% RSLogix 500 project VA116_TR_D.RSS, saved by version 7.10.00.09 %
PROJECT "VA116"    % processor: SLC 500, 1747-L532; 601760_CO2 %

PROGRAM FILES
  LAD 2 "601760_CO2"  66 rungs
  LAD 3 "INIT_ZAPN"  24 rungs
  LAD 4 "CASOVACE"  76 rungs
  LAD 5 "DIAGN_SPOL"  16 rungs
  LAD 6 "DIAGN_AUT"  98 rungs
  LAD 7 "DIAGN_K_VP"  28 rungs
  LAD 8 "HYDR_AGREG"  13 rungs
  LAD 9 "VODA_POHON"  16 rungs
  LAD 10 "REZIM_SER"  50 rungs
  LAD 11 "REZIM_RUC"  66 rungs
  LAD 12 "REZIM_VP"  18 rungs
  LAD 13 "REZIM_AUT"  28 rungs
  LAD 14 "REZIM_NULA"  6 rungs
  LAD 15 "STARTSTOP"  28 rungs
  LAD 16 "ZAKL_MECH"  92 rungs
  LAD 17 "KOPYTO_SOL"  22 rungs
  LAD 18 "HLAVA_SOLO"  23 rungs
  LAD 19 "KOPY_HLAVA"  37 rungs
  LAD 20 "STABILIZ"  24 rungs
  LAD 21 "ODDEL_IMP"  19 rungs
  LAD 22 "ODDEL_RS"  29 rungs
  LAD 23 "PODPUR_VZD"  17 rungs
  LAD 24 "VYFUK_TRN"  33 rungs
  LAD 25 "CO2"  8 rungs
  LAD 26 "VYSTUPY"  81 rungs
  LAD 27 "REC_ARCHIV"  4 rungs
  LAD 28 "REC_SAVE"  3 rungs
  LAD 29 "REC_LOAD"  4 rungs
  LAD 30 "REG_TEPLOT"  149 rungs

DATA FILES
  O0   38 elements
  I1   36 elements
  S2   83 elements
  B3   2 elements
  T4   82 elements
  C5   6 elements
  R6   1 elements
  N7   98 elements
  F8 FLOAT  10 elements
  N9   12 elements
  N10   256 elements
  N11   256 elements
  N12 N12  240 elements
  N13   255 elements
  N14   240 elements
  N15   240 elements

LADDER 2 "601760_CO2"
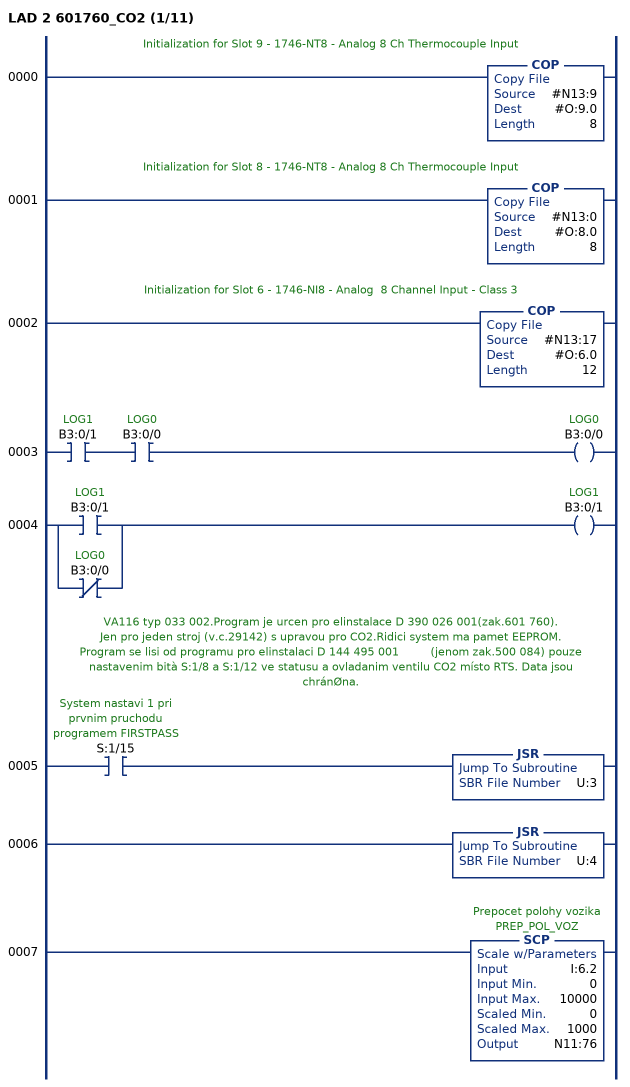
% Rung: 0 %
% Initialization for Slot 9 - 1746-NT8 - Analog 8 Ch Thermocouple Input %
SOR COP #N13:9 #O:9.0 8 EOR
% Rung: 1 %
% Initialization for Slot 8 - 1746-NT8 - Analog 8 Ch Thermocouple Input %
SOR COP #N13:0 #O:8.0 8 EOR
% Rung: 2 %
% Initialization for Slot 6 - 1746-NI8 - Analog  8 Channel Input - Class 3 %
SOR COP #N13:17 #O:6.0 12 EOR
% Rung: 3 %
SOR XIC B3:0/1 XIC B3:0/0 OTE B3:0/0 EOR
%   B3:0/1  LOG1 %
%   B3:0/0  LOG0 %
% Rung: 4 %
SOR BST XIC B3:0/1 NXB XIO B3:0/0 BND OTE B3:0/1 EOR
%   B3:0/1  LOG1 %
%   B3:0/0  LOG0 %
% Rung: 5 %
% VA116 typ 033 002.Program je urcen pro elinstalace D 390 026 001(zak.601 760).
% Jen pro jeden stroj (v.c.29142) s upravou pro CO2.Ridici system ma pamet EEPROM. Program se lisi od programu pro elinstalaci D 144 495 001         (jenom zak.500 084) pouze nastavenim bità S:1/8 a S:1/12 ve statusu a ovladanim ventilu CO2 místo RTS. Data jsou chránØna. %
SOR XIC S:1/15 JSR U:3 EOR
%   S:1/15  FIRSTPASS  "System nastavi 1 pri prvnim pruchodu programem" %
%   JSR U:3  "Iniciali- zace po zapnuti ridiciho systemu" %
% Rung: 6 %
SOR JSR U:4 EOR
%   JSR U:4  "Casovace, citace" %
% Rung: 7 %
SOR SCP I:6.2 0 10000 0 1000 N11:76 EOR
%   I:6.2  POL_VOZIKA  "Poloha vozika" %
%   N11:76  PREP_POL_VOZ  "Prepocet polohy vozika" %

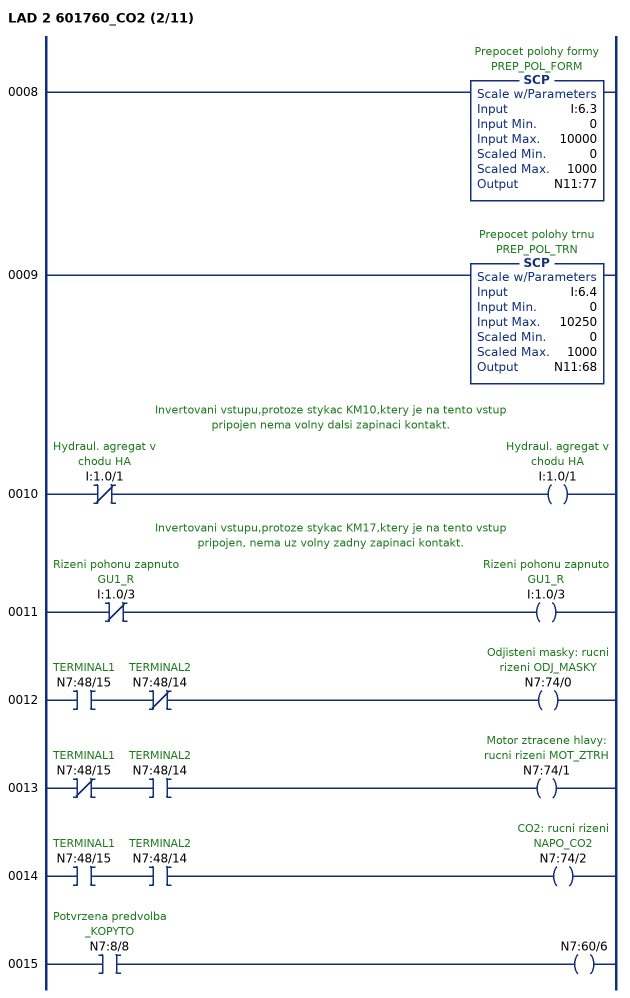
% Rung: 8 %
SOR SCP I:6.3 0 10000 0 1000 N11:77 EOR
%   I:6.3  POL_FORMY  "Poloha formy" %
%   N11:77  PREP_POL_FORM  "Prepocet polohy formy" %
% Rung: 9 %
SOR SCP I:6.4 0 10250 0 1000 N11:68 EOR
%   I:6.4  POL_VYF_TRNU  "Poloha vyfukovaciho trnu" %
%   N11:68  PREP_POL_TRN  "Prepocet polohy trnu" %
% Rung: 10 %
%         Invertovani vstupu,protoze stykac KM10,ktery je na tento vstup
%         pripojen nema volny dalsi zapinaci kontakt. %
SOR XIO I:1.0/1 OTE I:1.0/1 EOR
%   I:1.0/1  HA  "Hydraul. agregat v chodu" %
% Rung: 11 %
%          Invertovani vstupu,protoze stykac KM17,ktery je na tento vstup
%          pripojen, nema uz volny zadny zapinaci kontakt. %
SOR XIO I:1.0/3 OTE I:1.0/3 EOR
%   I:1.0/3  GU1_R  "Rizeni pohonu zapnuto" %
% Rung: 12 %
SOR XIC N7:48/15 XIO N7:48/14 OTE N7:74/0 EOR
%   N7:48/15  TERMINAL1 %
%   N7:48/14  TERMINAL2 %
%   N7:74/0  ODJ_MASKY  "Odjisteni masky: rucni rizeni" %
% Rung: 13 %
SOR XIO N7:48/15 XIC N7:48/14 OTE N7:74/1 EOR
%   N7:48/15  TERMINAL1 %
%   N7:48/14  TERMINAL2 %
%   N7:74/1  MOT_ZTRH  "Motor ztracene hlavy: rucni rizeni" %
% Rung: 14 %
SOR XIC N7:48/15 XIC N7:48/14 OTE N7:74/2 EOR
%   N7:48/15  TERMINAL1 %
%   N7:48/14  TERMINAL2 %
%   N7:74/2  NAPO_CO2  "CO2: rucni rizeni" %
% Rung: 15 %
SOR XIC N7:8/8 OTE N7:60/6 EOR
%   N7:8/8  _KOPYTO  "Potvrzena predvolba" %

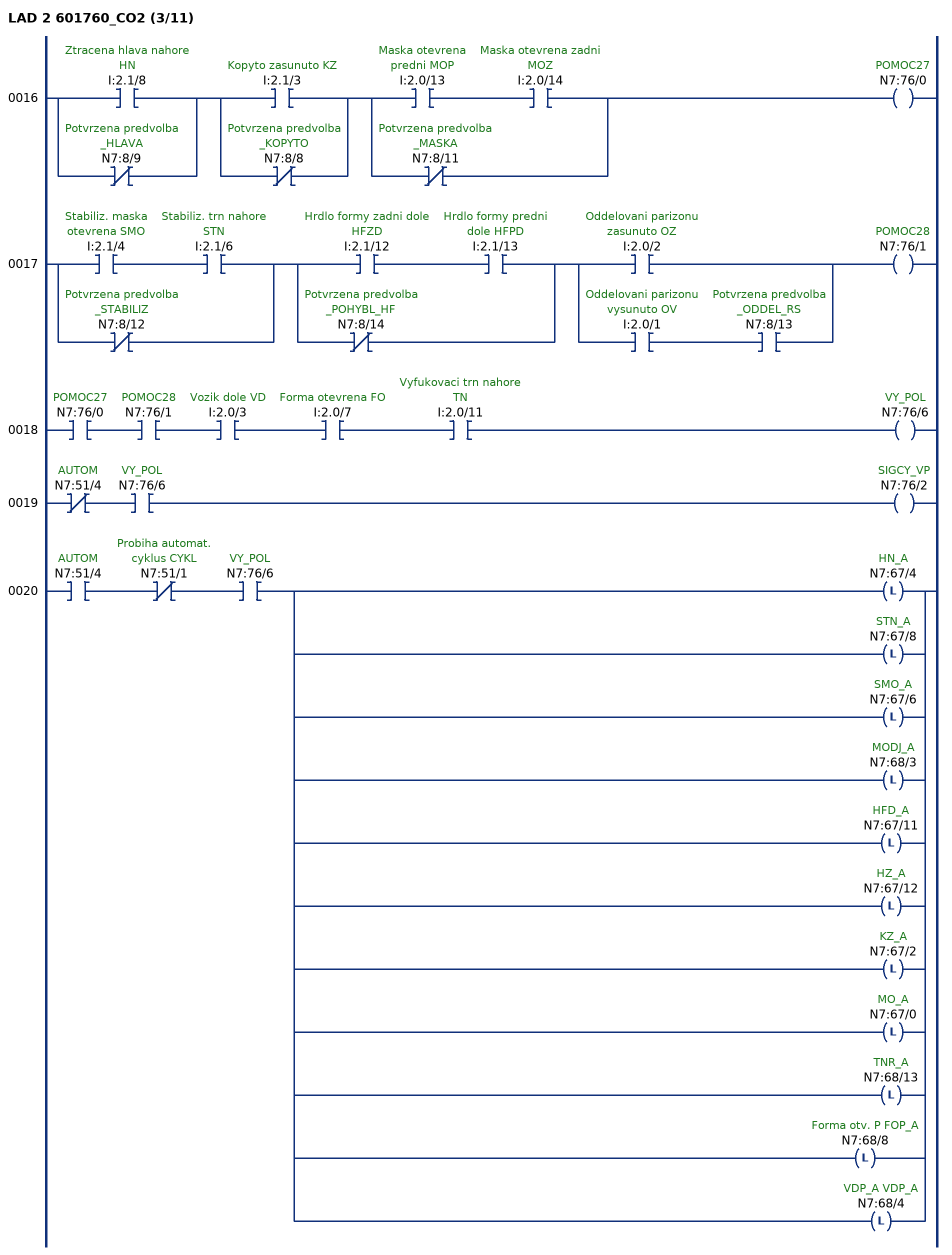
% Rung: 16 %
SOR BST XIC I:2.1/8 NXB XIO N7:8/9 BND BST XIC I:2.1/3 NXB XIO N7:8/8 BND BST XIC I:2.0/13 XIC I:2.0/14 NXB XIO N7:8/11 BND OTE N7:76/0 EOR
%   I:2.1/8  HN  "Ztracena hlava nahore" %
%   N7:8/9  _HLAVA  "Potvrzena predvolba" %
%   I:2.1/3  KZ  "Kopyto zasunuto" %
%   N7:8/8  _KOPYTO  "Potvrzena predvolba" %
%   I:2.0/13  MOP  "Maska otevrena predni" %
%   I:2.0/14  MOZ  "Maska otevrena zadni" %
%   N7:8/11  _MASKA  "Potvrzena predvolba" %
%   N7:76/0  POMOC27 %
% Rung: 17 %
SOR BST XIC I:2.1/4 XIC I:2.1/6 NXB XIO N7:8/12 BND BST XIC I:2.1/12 XIC I:2.1/13 NXB XIO N7:8/14 BND BST XIC I:2.0/2 NXB XIC I:2.0/1 XIC N7:8/13 BND OTE N7:76/1 EOR
%   I:2.1/4  SMO  "Stabiliz. maska otevrena" %
%   I:2.1/6  STN  "Stabiliz. trn nahore" %
%   N7:8/12  _STABILIZ  "Potvrzena predvolba" %
%   I:2.1/12  HFZD  "Hrdlo formy zadni dole" %
%   I:2.1/13  HFPD  "Hrdlo formy predni dole" %
%   N7:8/14  _POHYBL_HF  "Potvrzena predvolba" %
%   I:2.0/2  OZ  "Oddelovani parizonu zasunuto" %
%   I:2.0/1  OV  "Oddelovani parizonu vysunuto" %
%   N7:8/13  _ODDEL_RS  "Potvrzena predvolba" %
%   N7:76/1  POMOC28 %
% Rung: 18 %
SOR XIC N7:76/0 XIC N7:76/1 XIC I:2.0/3 XIC I:2.0/7 XIC I:2.0/11 OTE N7:76/6 EOR
%   N7:76/0  POMOC27 %
%   N7:76/1  POMOC28 %
%   I:2.0/3  VD  "Vozik dole" %
%   I:2.0/7  FO  "Forma otevrena" %
%   I:2.0/11  TN  "Vyfukovaci trn nahore" %
%   N7:76/6  VY_POL %
% Rung: 19 %
SOR XIO N7:51/4 XIC N7:76/6 OTE N7:76/2 EOR
%   N7:51/4  AUTOM %
%   N7:76/6  VY_POL %
%   N7:76/2  SIGCY_VP %
% Rung: 20 %
SOR XIC N7:51/4 XIO N7:51/1 XIC N7:76/6 BST OTL N7:67/4 NXB OTL N7:67/8 NXB OTL N7:67/6 NXB OTL N7:68/3 NXB OTL N7:67/11 NXB OTL N7:67/12 NXB OTL N7:67/2 NXB OTL N7:67/0 NXB OTL N7:68/13 NXB OTL N7:68/8 NXB OTL N7:68/4 BND EOR
%   N7:51/4  AUTOM %
%   N7:51/1  CYKL  "Probiha automat. cyklus" %
%   N7:76/6  VY_POL %
%   N7:67/4  HN_A %
%   N7:67/8  STN_A %
%   N7:67/6  SMO_A %
%   N7:68/3  MODJ_A %
%   N7:67/11  HFD_A %
%   N7:67/12  HZ_A %
%   N7:67/2  KZ_A %
%   N7:67/0  MO_A %
%   N7:68/13  TNR_A %
%   N7:68/8  FOP_A  "Forma otv. P" %
%   N7:68/4  VDP_A  "VDP_A" %

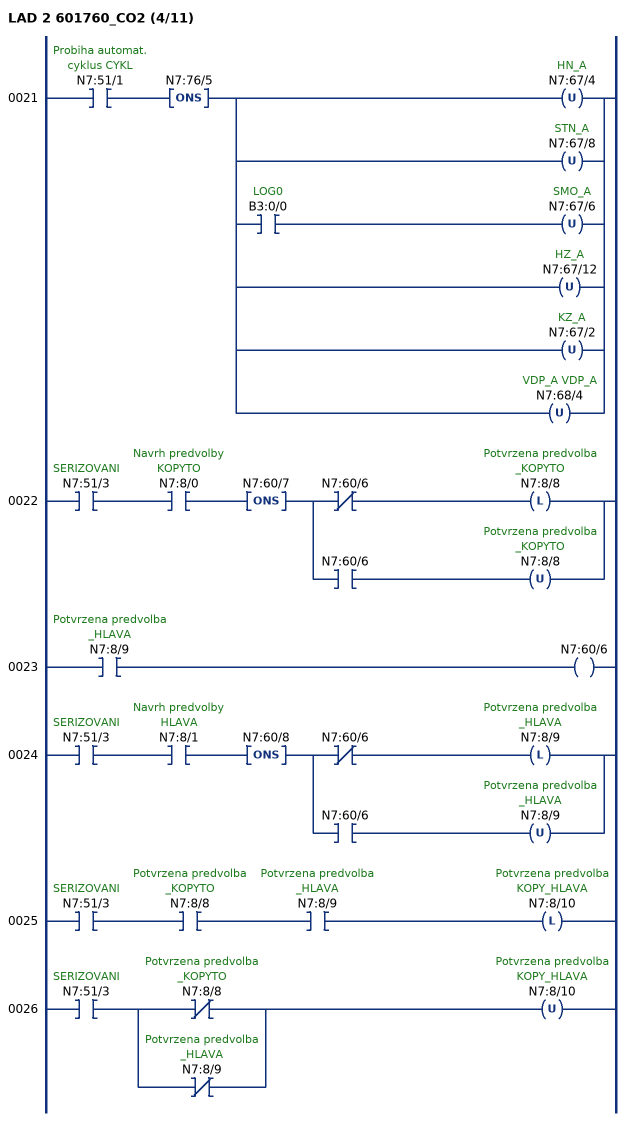
% Rung: 21 %
SOR XIC N7:51/1 OSR N7:76/5 BST OTU N7:67/4 NXB OTU N7:67/8 NXB XIC B3:0/0 OTU N7:67/6 NXB OTU N7:67/12 NXB OTU N7:67/2 NXB OTU N7:68/4 BND EOR
%   N7:51/1  CYKL  "Probiha automat. cyklus" %
%   N7:67/4  HN_A %
%   N7:67/8  STN_A %
%   B3:0/0  LOG0 %
%   N7:67/6  SMO_A %
%   N7:67/12  HZ_A %
%   N7:67/2  KZ_A %
%   N7:68/4  VDP_A  "VDP_A" %
% Rung: 22 %
SOR XIC N7:51/3 XIC N7:8/0 OSR N7:60/7 BST XIO N7:60/6 OTL N7:8/8 NXB XIC N7:60/6 OTU N7:8/8 BND EOR
%   N7:51/3  SERIZOVANI %
%   N7:8/0  KOPYTO  "Navrh predvolby" %
%   N7:8/8  _KOPYTO  "Potvrzena predvolba" %
% Rung: 23 %
SOR XIC N7:8/9 OTE N7:60/6 EOR
%   N7:8/9  _HLAVA  "Potvrzena predvolba" %
% Rung: 24 %
SOR XIC N7:51/3 XIC N7:8/1 OSR N7:60/8 BST XIO N7:60/6 OTL N7:8/9 NXB XIC N7:60/6 OTU N7:8/9 BND EOR
%   N7:51/3  SERIZOVANI %
%   N7:8/1  HLAVA  "Navrh predvolby" %
%   N7:8/9  _HLAVA  "Potvrzena predvolba" %
% Rung: 25 %
SOR XIC N7:51/3 XIC N7:8/8 XIC N7:8/9 OTL N7:8/10 EOR
%   N7:51/3  SERIZOVANI %
%   N7:8/8  _KOPYTO  "Potvrzena predvolba" %
%   N7:8/9  _HLAVA  "Potvrzena predvolba" %
%   N7:8/10  KOPY_HLAVA  "Potvrzena predvolba" %
% Rung: 26 %
SOR XIC N7:51/3 BST XIO N7:8/8 NXB XIO N7:8/9 BND OTU N7:8/10 EOR
%   N7:51/3  SERIZOVANI %
%   N7:8/8  _KOPYTO  "Potvrzena predvolba" %
%   N7:8/9  _HLAVA  "Potvrzena predvolba" %
%   N7:8/10  KOPY_HLAVA  "Potvrzena predvolba" %

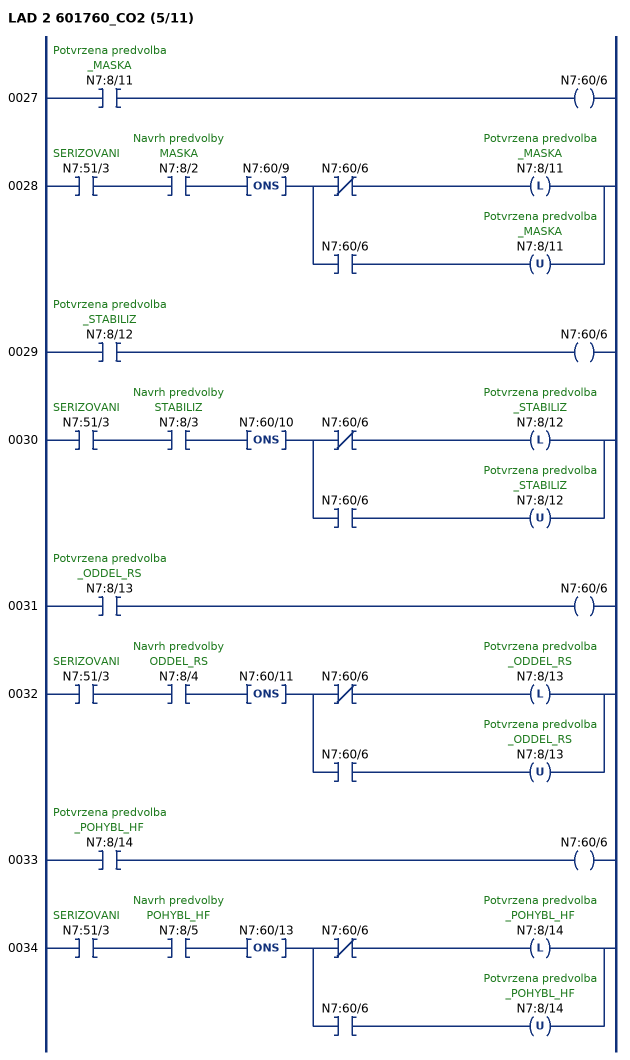
% Rung: 27 %
SOR XIC N7:8/11 OTE N7:60/6 EOR
%   N7:8/11  _MASKA  "Potvrzena predvolba" %
% Rung: 28 %
SOR XIC N7:51/3 XIC N7:8/2 OSR N7:60/9 BST XIO N7:60/6 OTL N7:8/11 NXB XIC N7:60/6 OTU N7:8/11 BND EOR
%   N7:51/3  SERIZOVANI %
%   N7:8/2  MASKA  "Navrh predvolby" %
%   N7:8/11  _MASKA  "Potvrzena predvolba" %
% Rung: 29 %
SOR XIC N7:8/12 OTE N7:60/6 EOR
%   N7:8/12  _STABILIZ  "Potvrzena predvolba" %
% Rung: 30 %
SOR XIC N7:51/3 XIC N7:8/3 OSR N7:60/10 BST XIO N7:60/6 OTL N7:8/12 NXB XIC N7:60/6 OTU N7:8/12 BND EOR
%   N7:51/3  SERIZOVANI %
%   N7:8/3  STABILIZ  "Navrh predvolby" %
%   N7:8/12  _STABILIZ  "Potvrzena predvolba" %
% Rung: 31 %
SOR XIC N7:8/13 OTE N7:60/6 EOR
%   N7:8/13  _ODDEL_RS  "Potvrzena predvolba" %
% Rung: 32 %
SOR XIC N7:51/3 XIC N7:8/4 OSR N7:60/11 BST XIO N7:60/6 OTL N7:8/13 NXB XIC N7:60/6 OTU N7:8/13 BND EOR
%   N7:51/3  SERIZOVANI %
%   N7:8/4  ODDEL_RS  "Navrh predvolby" %
%   N7:8/13  _ODDEL_RS  "Potvrzena predvolba" %
% Rung: 33 %
SOR XIC N7:8/14 OTE N7:60/6 EOR
%   N7:8/14  _POHYBL_HF  "Potvrzena predvolba" %
% Rung: 34 %
SOR XIC N7:51/3 XIC N7:8/5 OSR N7:60/13 BST XIO N7:60/6 OTL N7:8/14 NXB XIC N7:60/6 OTU N7:8/14 BND EOR
%   N7:51/3  SERIZOVANI %
%   N7:8/5  POHYBL_HF  "Navrh predvolby" %
%   N7:8/14  _POHYBL_HF  "Potvrzena predvolba" %

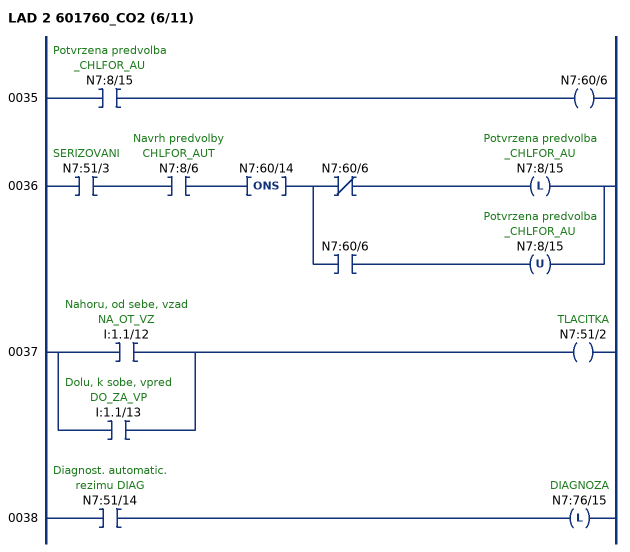
% Rung: 35 %
SOR XIC N7:8/15 OTE N7:60/6 EOR
%   N7:8/15  _CHLFOR_AU  "Potvrzena predvolba" %
% Rung: 36 %
SOR XIC N7:51/3 XIC N7:8/6 OSR N7:60/14 BST XIO N7:60/6 OTL N7:8/15 NXB XIC N7:60/6 OTU N7:8/15 BND EOR
%   N7:51/3  SERIZOVANI %
%   N7:8/6  CHLFOR_AUT  "Navrh predvolby" %
%   N7:8/15  _CHLFOR_AU  "Potvrzena predvolba" %
% Rung: 37 %
SOR BST XIC I:1.1/12 NXB XIC I:1.1/13 BND OTE N7:51/2 EOR
%   I:1.1/12  NA_OT_VZ  "Nahoru, od sebe, vzad" %
%   I:1.1/13  DO_ZA_VP  "Dolu, k sobe, vpred" %
%   N7:51/2  TLACITKA %
% Rung: 38 %
SOR XIC N7:51/14 OTL N7:76/15 EOR
%   N7:51/14  DIAG  "Diagnost. automatic. rezimu" %
%   N7:76/15  DIAGNOZA %

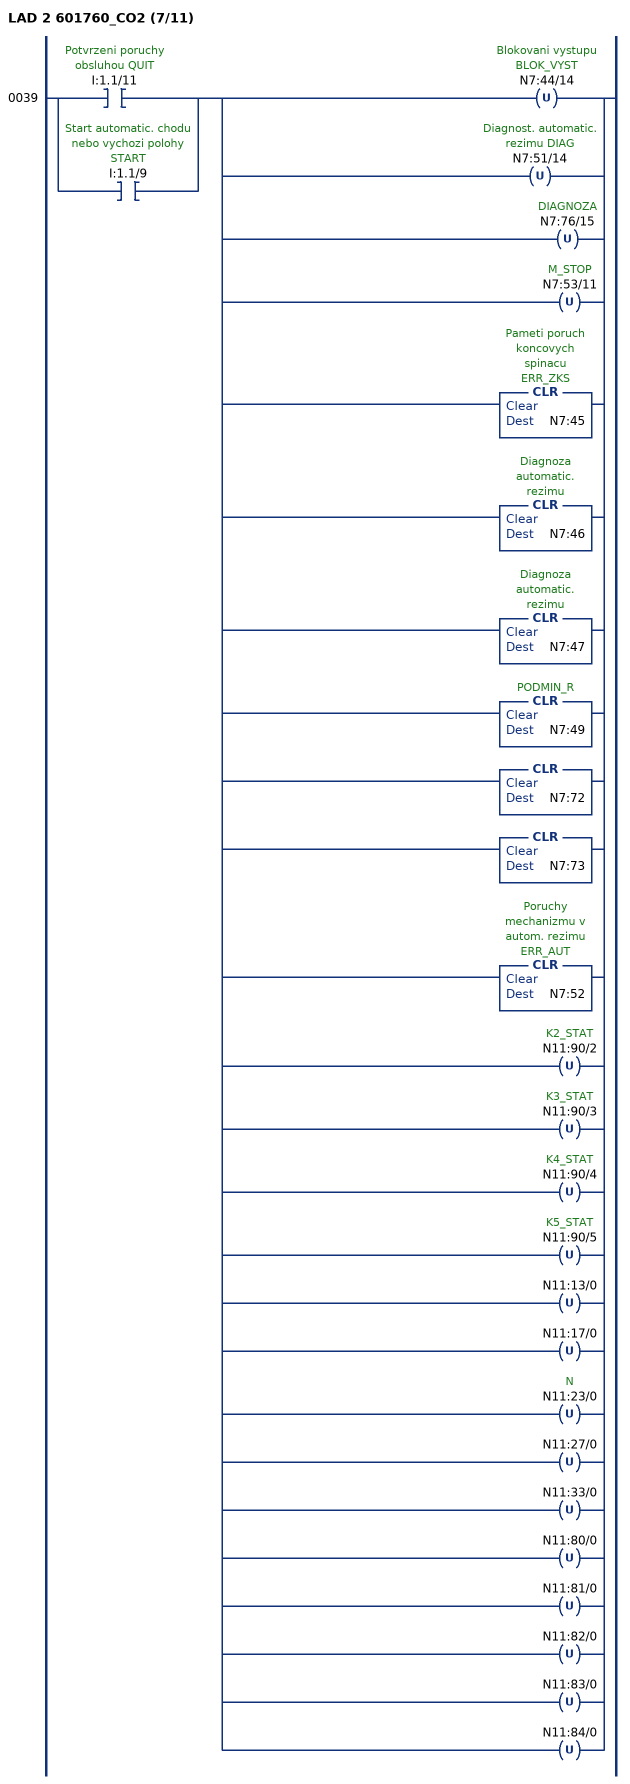
% Rung: 39 %
SOR BST XIC I:1.1/11 NXB XIC I:1.1/9 BND BST OTU N7:44/14 NXB OTU N7:51/14 NXB OTU N7:76/15 NXB OTU N7:53/11 NXB CLR N7:45 NXB CLR N7:46 NXB CLR N7:47 NXB CLR N7:49 NXB CLR N7:72 NXB CLR N7:73 NXB CLR N7:52 NXB OTU N11:90/2 NXB OTU N11:90/3 NXB OTU N11:90/4 NXB OTU N11:90/5 NXB OTU N11:13/0 NXB OTU N11:17/0 NXB OTU N11:23/0 NXB OTU N11:27/0 NXB OTU N11:33/0 NXB OTU N11:80/0 NXB OTU N11:81/0 NXB OTU N11:82/0 NXB OTU N11:83/0 NXB OTU N11:84/0 BND EOR
%   I:1.1/11  QUIT  "Potvrzeni poruchy obsluhou" %
%   I:1.1/9  START  "Start automatic. chodu nebo vychozi polohy" %
%   N7:44/14  BLOK_VYST  "Blokovani vystupu" %
%   N7:51/14  DIAG  "Diagnost. automatic. rezimu" %
%   N7:76/15  DIAGNOZA %
%   N7:53/11  M_STOP %
%   N7:45  ERR_ZKS  "Pameti poruch koncovych spinacu" %
%   N7:46  "Diagnoza automatic. rezimu" %
%   N7:47  "Diagnoza automatic. rezimu" %
%   N7:49  PODMIN_R %
%   CLR N7:49  "Podminky pro rucni rezim" %
%   N7:52  ERR_AUT  "Poruchy mechanizmu v autom. rezimu" %
%   N11:90/2  K2_STAT %
%   N11:90/3  K3_STAT %
%   N11:90/4  K4_STAT %
%   N11:90/5  K5_STAT %
%   N11:23/0  N %

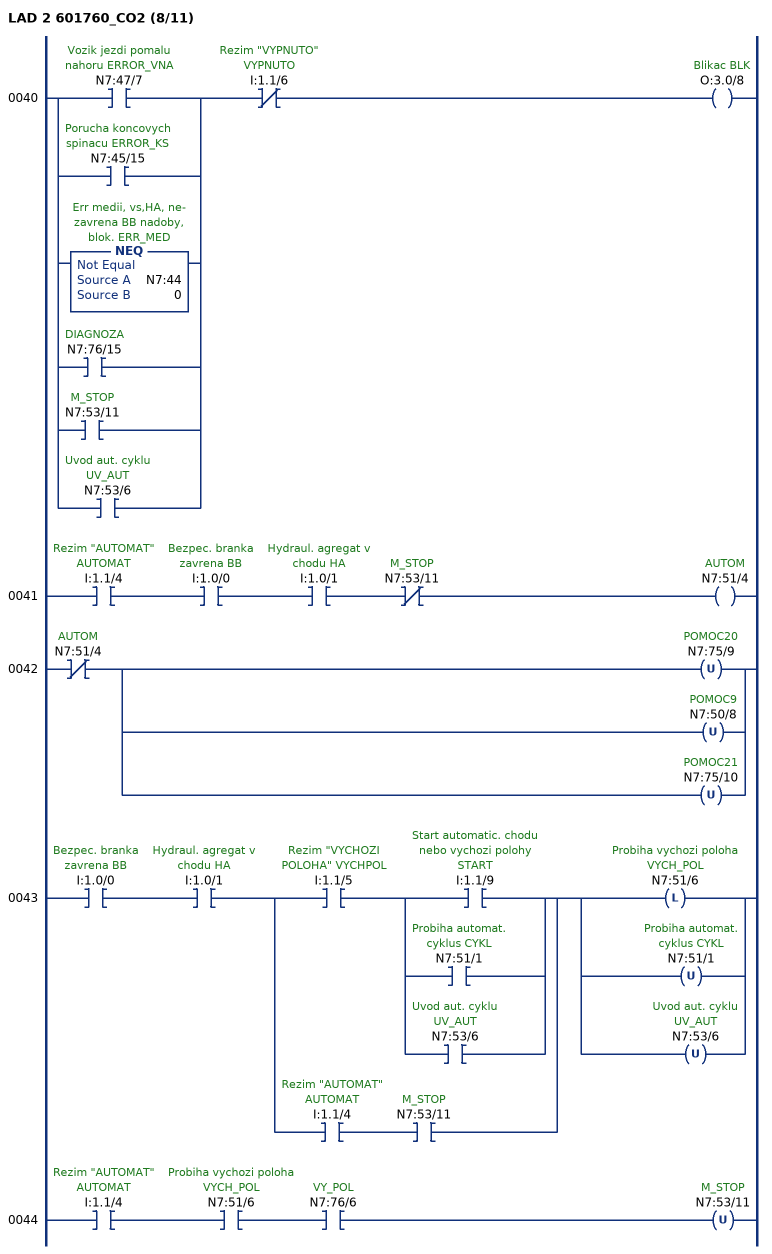
% Rung: 40 %
SOR BST XIC N7:47/7 NXB XIC N7:45/15 NXB NEQ N7:44 0 NXB XIC N7:76/15 NXB XIC N7:53/11 NXB XIC N7:53/6 BND XIO I:1.1/6 OTE O:3.0/8 EOR
%   N7:47/7  ERROR_VNA  "Vozik jezdi pomalu nahoru" %
%   N7:45/15  ERROR_KS  "Porucha koncovych spinacu" %
%   N7:44  ERR_MED  "Err medii, vs,HA, ne- zavrena BB nadoby, blok." %
%   N7:76/15  DIAGNOZA %
%   N7:53/11  M_STOP %
%   N7:53/6  UV_AUT  "Uvod aut. cyklu" %
%   I:1.1/6  VYPNUTO  "Rezim "VYPNUTO"" %
%   O:3.0/8  BLK  "Blikac" %
% Rung: 41 %
SOR XIC I:1.1/4 XIC I:1.0/0 XIC I:1.0/1 XIO N7:53/11 OTE N7:51/4 EOR
%   I:1.1/4  AUTOMAT  "Rezim "AUTOMAT"" %
%   I:1.0/0  BB  "Bezpec. branka zavrena" %
%   I:1.0/1  HA  "Hydraul. agregat v chodu" %
%   N7:53/11  M_STOP %
%   N7:51/4  AUTOM %
% Rung: 42 %
SOR XIO N7:51/4 BST OTU N7:75/9 NXB OTU N7:50/8 NXB OTU N7:75/10 BND EOR
%   N7:51/4  AUTOM %
%   N7:75/9  POMOC20 %
%   N7:50/8  POMOC9 %
%   N7:75/10  POMOC21 %
% Rung: 43 %
SOR XIC I:1.0/0 XIC I:1.0/1 BST XIC I:1.1/5 BST XIC I:1.1/9 NXB XIC N7:51/1 NXB XIC N7:53/6 BND NXB XIC I:1.1/4 XIC N7:53/11 BND BST OTL N7:51/6 NXB OTU N7:51/1 NXB OTU N7:53/6 BND EOR
%   I:1.0/0  BB  "Bezpec. branka zavrena" %
%   I:1.0/1  HA  "Hydraul. agregat v chodu" %
%   I:1.1/5  VYCHPOL  "Rezim "VYCHOZI POLOHA"" %
%   I:1.1/9  START  "Start automatic. chodu nebo vychozi polohy" %
%   N7:51/1  CYKL  "Probiha automat. cyklus" %
%   N7:53/6  UV_AUT  "Uvod aut. cyklu" %
%   I:1.1/4  AUTOMAT  "Rezim "AUTOMAT"" %
%   N7:53/11  M_STOP %
%   N7:51/6  VYCH_POL  "Probiha vychozi poloha" %
% Rung: 44 %
SOR XIC I:1.1/4 XIC N7:51/6 XIC N7:76/6 OTU N7:53/11 EOR
%   I:1.1/4  AUTOMAT  "Rezim "AUTOMAT"" %
%   N7:51/6  VYCH_POL  "Probiha vychozi poloha" %
%   N7:76/6  VY_POL %
%   N7:53/11  M_STOP %

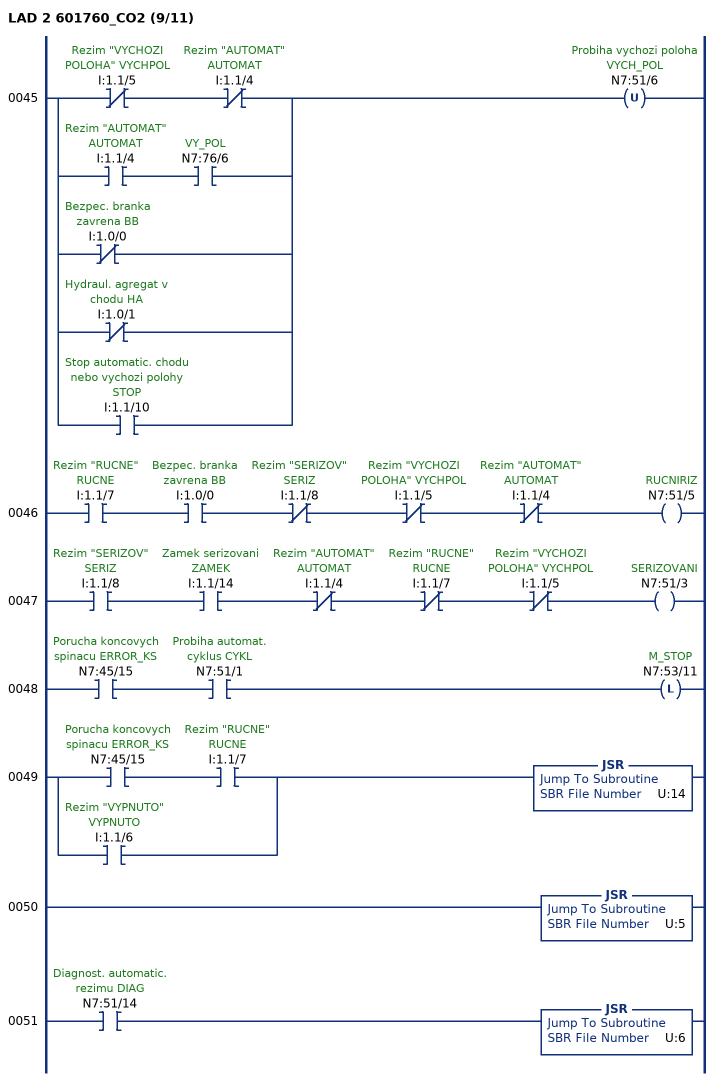
% Rung: 45 %
SOR BST XIO I:1.1/5 XIO I:1.1/4 NXB XIC I:1.1/4 XIC N7:76/6 NXB XIO I:1.0/0 NXB XIO I:1.0/1 NXB XIC I:1.1/10 BND OTU N7:51/6 EOR
%   I:1.1/5  VYCHPOL  "Rezim "VYCHOZI POLOHA"" %
%   I:1.1/4  AUTOMAT  "Rezim "AUTOMAT"" %
%   N7:76/6  VY_POL %
%   I:1.0/0  BB  "Bezpec. branka zavrena" %
%   I:1.0/1  HA  "Hydraul. agregat v chodu" %
%   I:1.1/10  STOP  "Stop automatic. chodu nebo vychozi polohy" %
%   N7:51/6  VYCH_POL  "Probiha vychozi poloha" %
% Rung: 46 %
SOR XIC I:1.1/7 XIC I:1.0/0 XIO I:1.1/8 XIO I:1.1/5 XIO I:1.1/4 OTE N7:51/5 EOR
%   I:1.1/7  RUCNE  "Rezim "RUCNE"" %
%   I:1.0/0  BB  "Bezpec. branka zavrena" %
%   I:1.1/8  SERIZ  "Rezim "SERIZOV"" %
%   I:1.1/5  VYCHPOL  "Rezim "VYCHOZI POLOHA"" %
%   I:1.1/4  AUTOMAT  "Rezim "AUTOMAT"" %
%   N7:51/5  RUCNIRIZ %
% Rung: 47 %
SOR XIC I:1.1/8 XIC I:1.1/14 XIO I:1.1/4 XIO I:1.1/7 XIO I:1.1/5 OTE N7:51/3 EOR
%   I:1.1/8  SERIZ  "Rezim "SERIZOV"" %
%   I:1.1/14  ZAMEK  "Zamek serizovani" %
%   I:1.1/4  AUTOMAT  "Rezim "AUTOMAT"" %
%   I:1.1/7  RUCNE  "Rezim "RUCNE"" %
%   I:1.1/5  VYCHPOL  "Rezim "VYCHOZI POLOHA"" %
%   N7:51/3  SERIZOVANI %
% Rung: 48 %
SOR XIC N7:45/15 XIC N7:51/1 OTL N7:53/11 EOR
%   N7:45/15  ERROR_KS  "Porucha koncovych spinacu" %
%   N7:51/1  CYKL  "Probiha automat. cyklus" %
%   N7:53/11  M_STOP %
% Rung: 49 %
SOR BST XIC N7:45/15 XIC I:1.1/7 NXB XIC I:1.1/6 BND JSR U:14 EOR
%   N7:45/15  ERROR_KS  "Porucha koncovych spinacu" %
%   I:1.1/7  RUCNE  "Rezim "RUCNE"" %
%   I:1.1/6  VYPNUTO  "Rezim "VYPNUTO"" %
%   JSR U:14  "Rezim VYPNUTO" %
% Rung: 50 %
SOR JSR U:5 EOR
%   JSR U:5  "Diagnosti- ka spolec- na pro vsechny rezimy" %
% Rung: 51 %
SOR XIC N7:51/14 JSR U:6 EOR
%   N7:51/14  DIAG  "Diagnost. automatic. rezimu" %
%   JSR U:6  "Diagnosti- ka zavad v automa- tickem rezimu" %

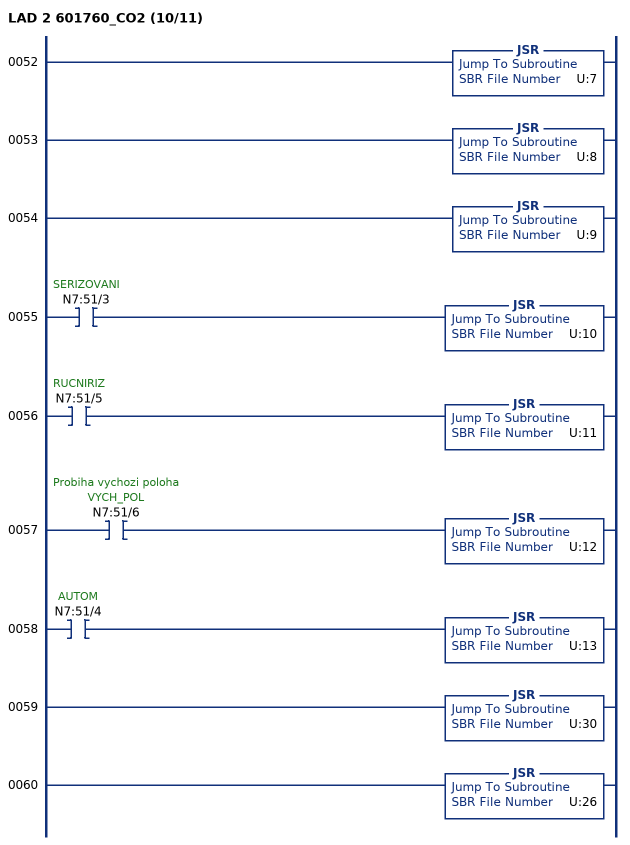
% Rung: 52 %
SOR JSR U:7 EOR
%   JSR U:7  "Hlidani prorazeni koncovych spinacu" %
% Rung: 53 %
SOR JSR U:8 EOR
%   JSR U:8  "Rizeni hydraul. agregatu" %
% Rung: 54 %
SOR JSR U:9 EOR
%   JSR U:9  "Chlazeni formy vodou, pohon VS" %
% Rung: 55 %
SOR XIC N7:51/3 JSR U:10 EOR
%   N7:51/3  SERIZOVANI %
%   JSR U:10  "Rezim SERIZOVANI" %
% Rung: 56 %
SOR XIC N7:51/5 JSR U:11 EOR
%   N7:51/5  RUCNIRIZ %
%   JSR U:11  "Rezim RUCNE" %
% Rung: 57 %
SOR XIC N7:51/6 JSR U:12 EOR
%   N7:51/6  VYCH_POL  "Probiha vychozi poloha" %
%   JSR U:12  "Rezim VYCHOZI POLOHA" %
% Rung: 58 %
SOR XIC N7:51/4 JSR U:13 EOR
%   N7:51/4  AUTOM %
%   JSR U:13  "Rezim AUTOMAT" %
% Rung: 59 %
SOR JSR U:30 EOR
% Rung: 60 %
SOR JSR U:26 EOR
%   JSR U:26  "VYSTUPY" %

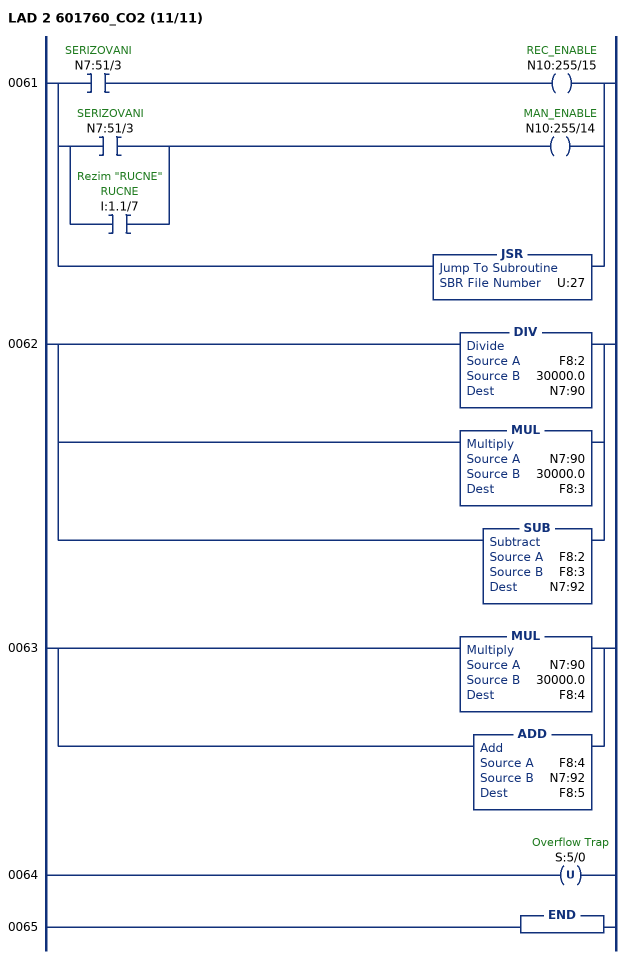
% Rung: 61 %
SOR BST XIC N7:51/3 OTE N10:255/15 NXB BST XIC N7:51/3 NXB XIC I:1.1/7 BND OTE N10:255/14 NXB JSR U:27 BND EOR
%   N7:51/3  SERIZOVANI %
%   N10:255/15  REC_ENABLE %
%   I:1.1/7  RUCNE  "Rezim "RUCNE"" %
%   N10:255/14  MAN_ENABLE %
%   JSR U:27  "Archivace receptur" %
% Rung: 62 %
SOR BST DIV F8:2 30000.0 N7:90 NXB MUL N7:90 30000.0 F8:3 NXB SUB F8:2 F8:3 N7:92 BND EOR
% Rung: 63 %
SOR BST MUL N7:90 30000.0 F8:4 NXB ADD F8:4 N7:92 F8:5 BND EOR
% Rung: 64 %
SOR OTU S:5/0 EOR
%   S:5/0  "Overflow Trap" %
% Rung: 65 %
SOR END EOR

LADDER 3 "INIT_ZAPN"
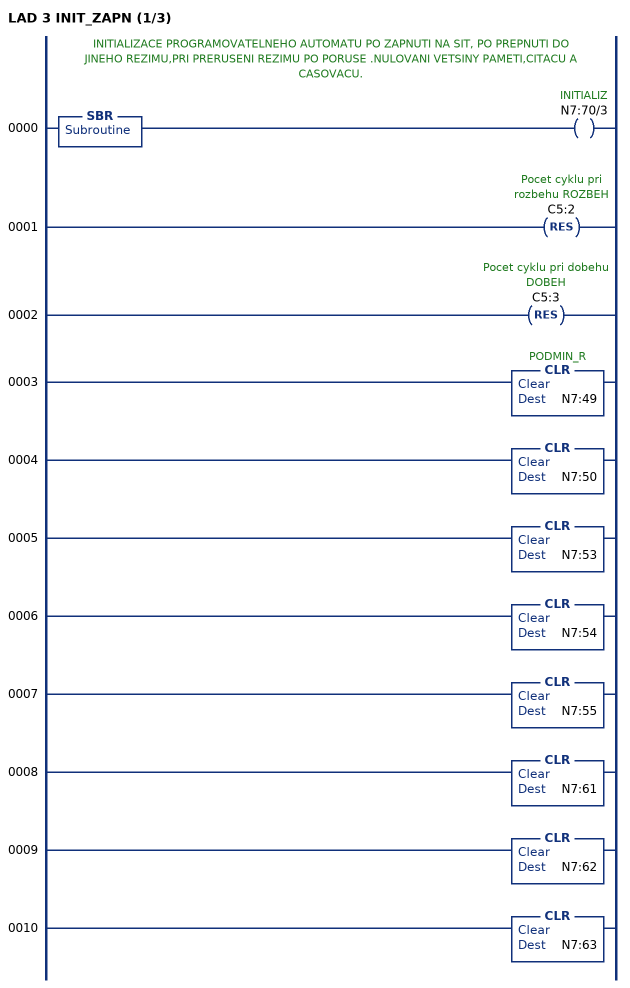
% Rung: 0 %
% INITIALIZACE PROGRAMOVATELNEHO AUTOMATU PO ZAPNUTI NA SIT, PO PREPNUTI DO  JINEHO REZIMU,PRI PRERUSENI REZIMU PO PORUSE .NULOVANI VETSINY PAMETI,CITACU A CASOVACU. %
SOR SBR OTE N7:70/3 EOR
%   N7:70/3  INITIALIZ %
% Rung: 1 %
SOR RES C5:2 EOR
%   C5:2  ROZBEH  "Pocet cyklu pri rozbehu" %
% Rung: 2 %
SOR RES C5:3 EOR
%   C5:3  DOBEH  "Pocet cyklu pri dobehu" %
% Rung: 3 %
SOR CLR N7:49 EOR
%   N7:49  PODMIN_R %
%   CLR N7:49  "Podminky pro rucni rezim" %
% Rung: 4 %
SOR CLR N7:50 EOR
%   CLR N7:50  "Pomocne merkry" %
% Rung: 5 %
SOR CLR N7:53 EOR
%   CLR N7:53  "Pameti automatic. rezimu" %
% Rung: 6 %
SOR CLR N7:54 EOR
%   CLR N7:54  "Logicke operandy casovacu" %
% Rung: 7 %
SOR CLR N7:55 EOR
%   CLR N7:55  "Logicke operandy casovacu" %
% Rung: 8 %
SOR CLR N7:61 EOR
%   CLR N7:61  "Pameti automatic. rezimu" %
% Rung: 9 %
SOR CLR N7:62 EOR
%   CLR N7:62  "Merkry vystupu vychozi polohy" %
% Rung: 10 %
SOR CLR N7:63 EOR
%   CLR N7:63  "Merkry vystupu rucniho rezimu" %

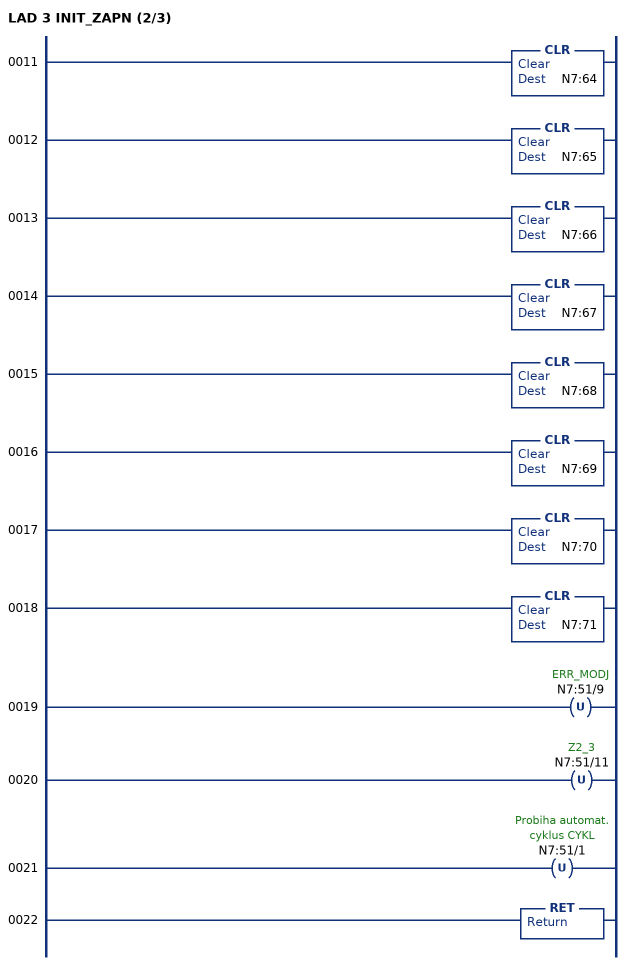
% Rung: 11 %
SOR CLR N7:64 EOR
%   CLR N7:64  "Merkry vystupu rucniho rezimu" %
% Rung: 12 %
SOR CLR N7:65 EOR
%   CLR N7:65  "Merkry vystupu rezimu serizovani" %
% Rung: 13 %
SOR CLR N7:66 EOR
%   CLR N7:66  "Merkry vystupu rezimu serizovani" %
% Rung: 14 %
SOR CLR N7:67 EOR
%   CLR N7:67  "Merkry vystupu automatic. rezimu" %
% Rung: 15 %
SOR CLR N7:68 EOR
%   CLR N7:68  "Merkry vystupu automatic. rezimu" %
% Rung: 16 %
SOR CLR N7:69 EOR
%   CLR N7:69  "Merkry vystupu automatic. rezimu, rampy" %
% Rung: 17 %
SOR CLR N7:70 EOR
%   CLR N7:70  "Zacatky failu" %
% Rung: 18 %
SOR CLR N7:71 EOR
%   CLR N7:71  "Zacatky failu" %
% Rung: 19 %
SOR OTU N7:51/9 EOR
%   N7:51/9  ERR_MODJ %
% Rung: 20 %
SOR OTU N7:51/11 EOR
%   N7:51/11  Z2_3 %
% Rung: 21 %
SOR OTU N7:51/1 EOR
%   N7:51/1  CYKL  "Probiha automat. cyklus" %
% Rung: 22 %
SOR RET EOR

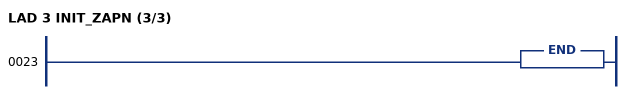
% Rung: 23 %
SOR END EOR

LADDER 4 "CASOVACE"
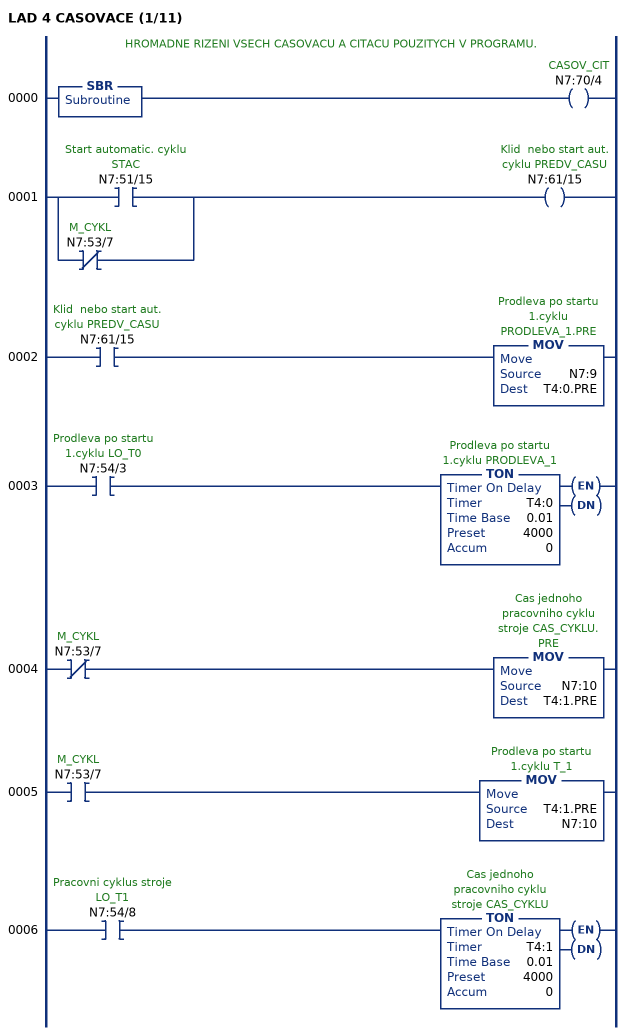
% Rung: 0 %
% HROMADNE RIZENI VSECH CASOVACU A CITACU POUZITYCH V PROGRAMU. %
SOR SBR OTE N7:70/4 EOR
%   N7:70/4  CASOV_CIT %
% Rung: 1 %
SOR BST XIC N7:51/15 NXB XIO N7:53/7 BND OTE N7:61/15 EOR
%   N7:51/15  STAC  "Start automatic. cyklu" %
%   N7:53/7  M_CYKL %
%   N7:61/15  PREDV_CASU  "Klid  nebo start aut. cyklu" %
% Rung: 2 %
SOR XIC N7:61/15 MOV N7:9 T4:0.PRE EOR
%   N7:61/15  PREDV_CASU  "Klid  nebo start aut. cyklu" %
%   N7:9  T_0  "Pracovni cyklus stroje" %
%   T4:0  PRODLEVA_1  "Prodleva po startu 1.cyklu" %
% Rung: 3 %
SOR XIC N7:54/3 TON T4:0 0.01 4000 0 EOR
%   N7:54/3  LO_T0  "Prodleva po startu 1.cyklu" %
%   T4:0  PRODLEVA_1  "Prodleva po startu 1.cyklu" %
% Rung: 4 %
SOR XIO N7:53/7 MOV N7:10 T4:1.PRE EOR
%   N7:53/7  M_CYKL %
%   N7:10  T_1  "Prodleva po startu 1.cyklu" %
%   T4:1  CAS_CYKLU  "Cas jednoho pracovniho cyklu stroje" %
% Rung: 5 %
SOR XIC N7:53/7 MOV T4:1.PRE N7:10 EOR
%   N7:53/7  M_CYKL %
%   T4:1  CAS_CYKLU  "Cas jednoho pracovniho cyklu stroje" %
%   N7:10  T_1  "Prodleva po startu 1.cyklu" %
% Rung: 6 %
SOR XIC N7:54/8 TON T4:1 0.01 4000 0 EOR
%   N7:54/8  LO_T1  "Pracovni cyklus stroje" %
%   T4:1  CAS_CYKLU  "Cas jednoho pracovniho cyklu stroje" %

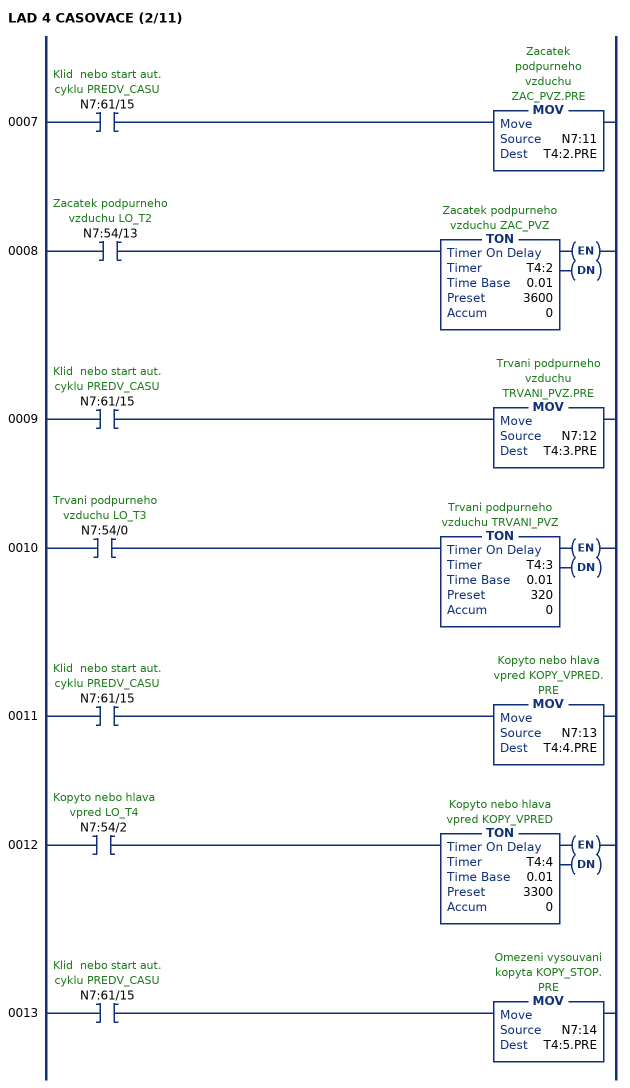
% Rung: 7 %
SOR XIC N7:61/15 MOV N7:11 T4:2.PRE EOR
%   N7:61/15  PREDV_CASU  "Klid  nebo start aut. cyklu" %
%   N7:11  T_2  "Zacatek podpurneho vzduchu" %
%   T4:2  ZAC_PVZ  "Zacatek podpurneho vzduchu" %
% Rung: 8 %
SOR XIC N7:54/13 TON T4:2 0.01 3600 0 EOR
%   N7:54/13  LO_T2  "Zacatek podpurneho vzduchu" %
%   T4:2  ZAC_PVZ  "Zacatek podpurneho vzduchu" %
% Rung: 9 %
SOR XIC N7:61/15 MOV N7:12 T4:3.PRE EOR
%   N7:61/15  PREDV_CASU  "Klid  nebo start aut. cyklu" %
%   N7:12  T_3  "Trvani podpurneho vzduchu" %
%   T4:3  TRVANI_PVZ  "Trvani podpurneho vzduchu" %
% Rung: 10 %
SOR XIC N7:54/0 TON T4:3 0.01 320 0 EOR
%   N7:54/0  LO_T3  "Trvani podpurneho vzduchu" %
%   T4:3  TRVANI_PVZ  "Trvani podpurneho vzduchu" %
% Rung: 11 %
SOR XIC N7:61/15 MOV N7:13 T4:4.PRE EOR
%   N7:61/15  PREDV_CASU  "Klid  nebo start aut. cyklu" %
%   N7:13  T_4  "Kopyto nebo hlava vpred" %
%   T4:4  KOPY_VPRED  "Kopyto nebo hlava vpred" %
% Rung: 12 %
SOR XIC N7:54/2 TON T4:4 0.01 3300 0 EOR
%   N7:54/2  LO_T4  "Kopyto nebo hlava vpred" %
%   T4:4  KOPY_VPRED  "Kopyto nebo hlava vpred" %
% Rung: 13 %
SOR XIC N7:61/15 MOV N7:14 T4:5.PRE EOR
%   N7:61/15  PREDV_CASU  "Klid  nebo start aut. cyklu" %
%   N7:14  T_5  "Omezeni vysouvani kopyta" %
%   T4:5  KOPY_STOP  "Omezeni vysouvani kopyta" %

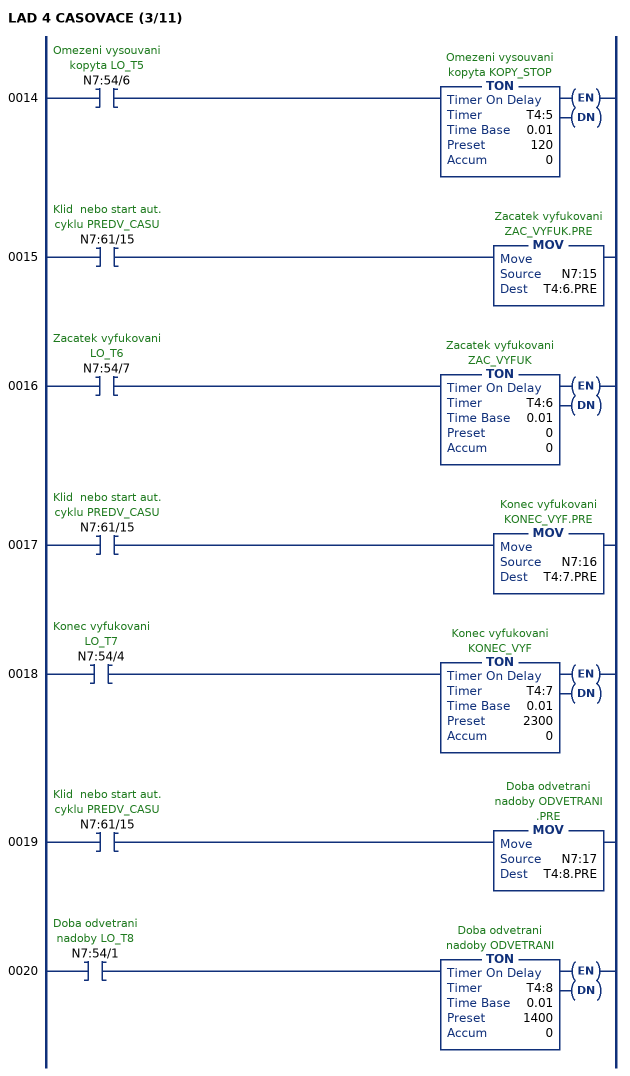
% Rung: 14 %
SOR XIC N7:54/6 TON T4:5 0.01 120 0 EOR
%   N7:54/6  LO_T5  "Omezeni vysouvani kopyta" %
%   T4:5  KOPY_STOP  "Omezeni vysouvani kopyta" %
% Rung: 15 %
SOR XIC N7:61/15 MOV N7:15 T4:6.PRE EOR
%   N7:61/15  PREDV_CASU  "Klid  nebo start aut. cyklu" %
%   N7:15  T_6  "Zacatek vyfukovani" %
%   T4:6  ZAC_VYFUK  "Zacatek vyfukovani" %
% Rung: 16 %
SOR XIC N7:54/7 TON T4:6 0.01 0 0 EOR
%   N7:54/7  LO_T6  "Zacatek vyfukovani" %
%   T4:6  ZAC_VYFUK  "Zacatek vyfukovani" %
% Rung: 17 %
SOR XIC N7:61/15 MOV N7:16 T4:7.PRE EOR
%   N7:61/15  PREDV_CASU  "Klid  nebo start aut. cyklu" %
%   N7:16  T_7  "Konec vyfukovani" %
%   T4:7  KONEC_VYF  "Konec vyfukovani" %
% Rung: 18 %
SOR XIC N7:54/4 TON T4:7 0.01 2300 0 EOR
%   N7:54/4  LO_T7  "Konec vyfukovani" %
%   T4:7  KONEC_VYF  "Konec vyfukovani" %
% Rung: 19 %
SOR XIC N7:61/15 MOV N7:17 T4:8.PRE EOR
%   N7:61/15  PREDV_CASU  "Klid  nebo start aut. cyklu" %
%   N7:17  T_8  "Doba odvetrani nadoby" %
%   T4:8  ODVETRANI  "Doba odvetrani nadoby" %
% Rung: 20 %
SOR XIC N7:54/1 TON T4:8 0.01 1400 0 EOR
%   N7:54/1  LO_T8  "Doba odvetrani nadoby" %
%   T4:8  ODVETRANI  "Doba odvetrani nadoby" %

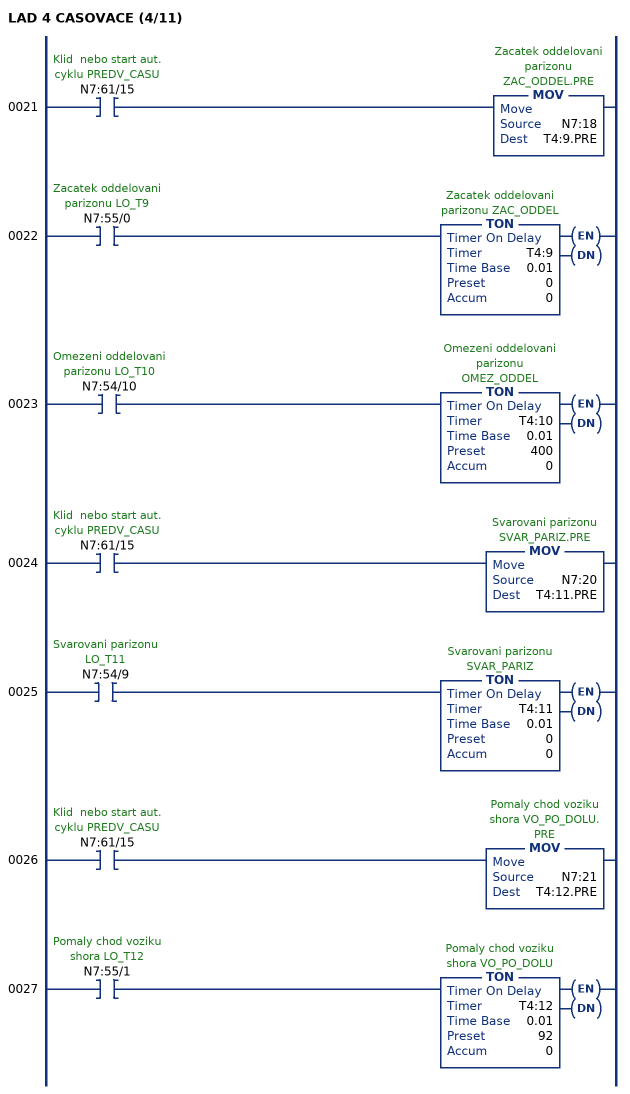
% Rung: 21 %
SOR XIC N7:61/15 MOV N7:18 T4:9.PRE EOR
%   N7:61/15  PREDV_CASU  "Klid  nebo start aut. cyklu" %
%   N7:18  T_9  "Zacatek oddelovani parizonu" %
%   T4:9  ZAC_ODDEL  "Zacatek oddelovani parizonu" %
% Rung: 22 %
SOR XIC N7:55/0 TON T4:9 0.01 0 0 EOR
%   N7:55/0  LO_T9  "Zacatek oddelovani parizonu" %
%   T4:9  ZAC_ODDEL  "Zacatek oddelovani parizonu" %
% Rung: 23 %
SOR XIC N7:54/10 TON T4:10 0.01 400 0 EOR
%   N7:54/10  LO_T10  "Omezeni oddelovani parizonu" %
%   T4:10  OMEZ_ODDEL  "Omezeni oddelovani parizonu" %
% Rung: 24 %
SOR XIC N7:61/15 MOV N7:20 T4:11.PRE EOR
%   N7:61/15  PREDV_CASU  "Klid  nebo start aut. cyklu" %
%   N7:20  T_11  "Svarovani parizonu" %
%   T4:11  SVAR_PARIZ  "Svarovani parizonu" %
% Rung: 25 %
SOR XIC N7:54/9 TON T4:11 0.01 0 0 EOR
%   N7:54/9  LO_T11  "Svarovani parizonu" %
%   T4:11  SVAR_PARIZ  "Svarovani parizonu" %
% Rung: 26 %
SOR XIC N7:61/15 MOV N7:21 T4:12.PRE EOR
%   N7:61/15  PREDV_CASU  "Klid  nebo start aut. cyklu" %
%   N7:21  T_12  "Pomaly chod voziku shora" %
%   T4:12  VO_PO_DOLU  "Pomaly chod voziku shora" %
% Rung: 27 %
SOR XIC N7:55/1 TON T4:12 0.01 92 0 EOR
%   N7:55/1  LO_T12  "Pomaly chod voziku shora" %
%   T4:12  VO_PO_DOLU  "Pomaly chod voziku shora" %

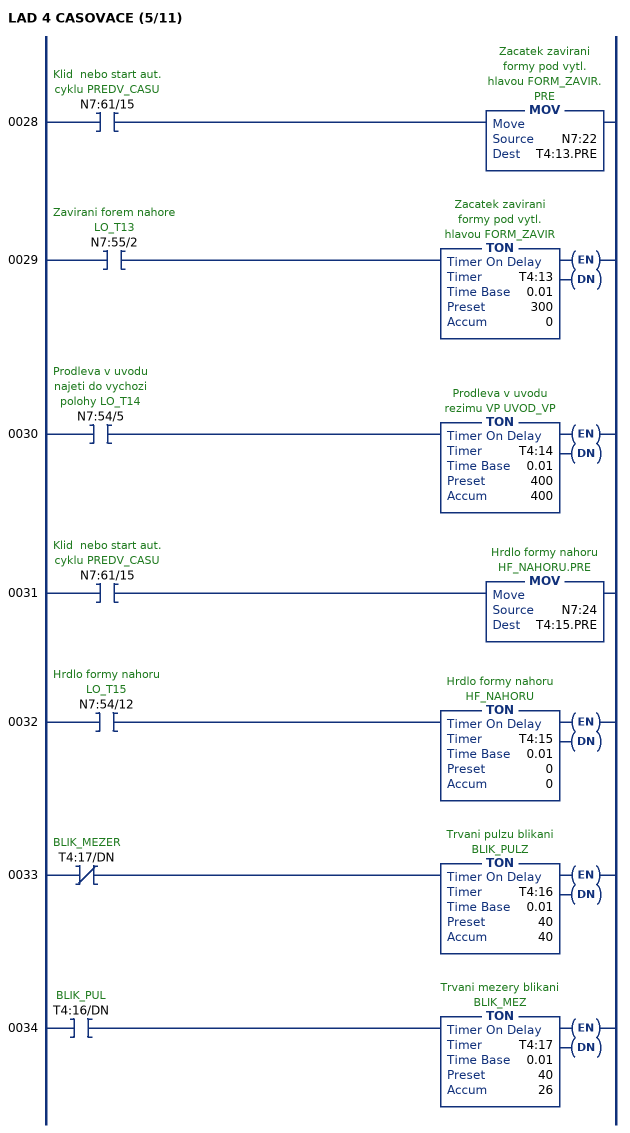
% Rung: 28 %
SOR XIC N7:61/15 MOV N7:22 T4:13.PRE EOR
%   N7:61/15  PREDV_CASU  "Klid  nebo start aut. cyklu" %
%   N7:22  T_13  "Zavirani forem nahore" %
%   T4:13  FORM_ZAVIR  "Zacatek zavirani formy pod vytl. hlavou" %
% Rung: 29 %
SOR XIC N7:55/2 TON T4:13 0.01 300 0 EOR
%   N7:55/2  LO_T13  "Zavirani forem nahore" %
%   T4:13  FORM_ZAVIR  "Zacatek zavirani formy pod vytl. hlavou" %
% Rung: 30 %
SOR XIC N7:54/5 TON T4:14 0.01 400 400 EOR
%   N7:54/5  LO_T14  "Prodleva v uvodu najeti do vychozi polohy" %
%   T4:14  UVOD_VP  "Prodleva v uvodu rezimu VP" %
% Rung: 31 %
SOR XIC N7:61/15 MOV N7:24 T4:15.PRE EOR
%   N7:61/15  PREDV_CASU  "Klid  nebo start aut. cyklu" %
%   N7:24  T_15  "Hrdlo formy nahoru" %
%   T4:15  HF_NAHORU  "Hrdlo formy nahoru" %
% Rung: 32 %
SOR XIC N7:54/12 TON T4:15 0.01 0 0 EOR
%   N7:54/12  LO_T15  "Hrdlo formy nahoru" %
%   T4:15  HF_NAHORU  "Hrdlo formy nahoru" %
% Rung: 33 %
SOR XIO T4:17/DN TON T4:16 0.01 40 40 EOR
%   T4:17/DN  BLIK_MEZER %
%   T4:16  BLIK_PULZ  "Trvani pulzu blikani" %
% Rung: 34 %
SOR XIC T4:16/DN TON T4:17 0.01 40 26 EOR
%   T4:16/DN  BLIK_PUL %
%   T4:17  BLIK_MEZ  "Trvani mezery blikani" %

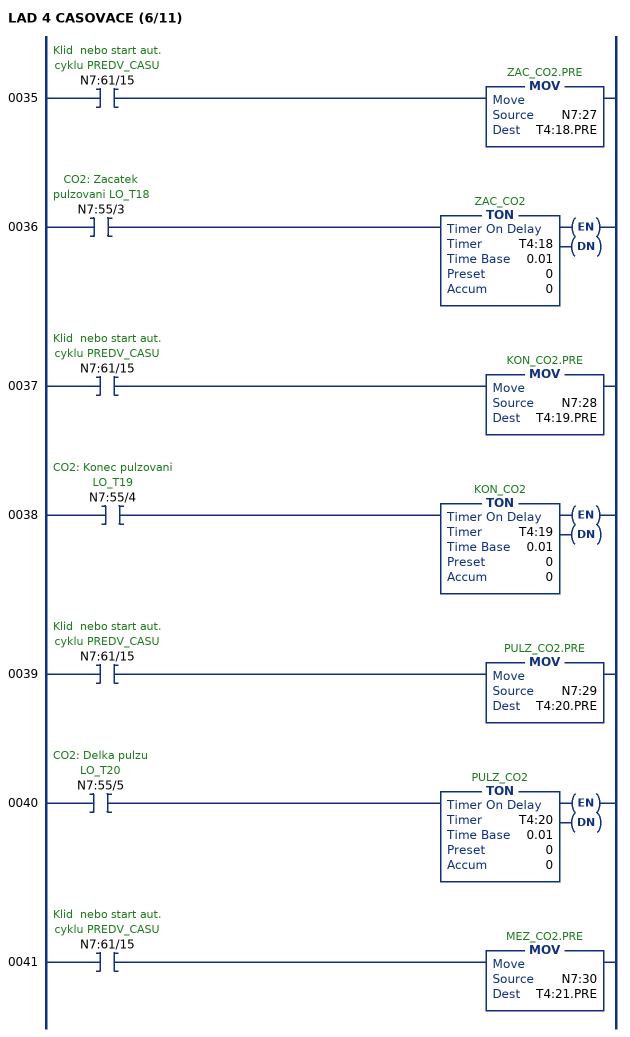
% Rung: 35 %
SOR XIC N7:61/15 MOV N7:27 T4:18.PRE EOR
%   N7:61/15  PREDV_CASU  "Klid  nebo start aut. cyklu" %
%   N7:27  T_18  "RTS: vytlacov. trn nahoru 1" %
%   T4:18  ZAC_CO2 %
% Rung: 36 %
SOR XIC N7:55/3 TON T4:18 0.01 0 0 EOR
%   N7:55/3  LO_T18  "CO2: Zacatek pulzovani" %
%   T4:18  ZAC_CO2 %
% Rung: 37 %
SOR XIC N7:61/15 MOV N7:28 T4:19.PRE EOR
%   N7:61/15  PREDV_CASU  "Klid  nebo start aut. cyklu" %
%   N7:28  T_19  "RTS: vytlacov. trn dolu 1" %
%   T4:19  KON_CO2 %
% Rung: 38 %
SOR XIC N7:55/4 TON T4:19 0.01 0 0 EOR
%   N7:55/4  LO_T19  "CO2: Konec pulzovani" %
%   T4:19  KON_CO2 %
% Rung: 39 %
SOR XIC N7:61/15 MOV N7:29 T4:20.PRE EOR
%   N7:61/15  PREDV_CASU  "Klid  nebo start aut. cyklu" %
%   N7:29  T_20  "RTS: vytlacov. trn nahoru 2" %
%   T4:20  PULZ_CO2 %
% Rung: 40 %
SOR XIC N7:55/5 TON T4:20 0.01 0 0 EOR
%   N7:55/5  LO_T20  "CO2: Delka pulzu" %
%   T4:20  PULZ_CO2 %
% Rung: 41 %
SOR XIC N7:61/15 MOV N7:30 T4:21.PRE EOR
%   N7:61/15  PREDV_CASU  "Klid  nebo start aut. cyklu" %
%   N7:30  T_21  "RTS: vytlacov. trn dolu 2" %
%   T4:21  MEZ_CO2 %

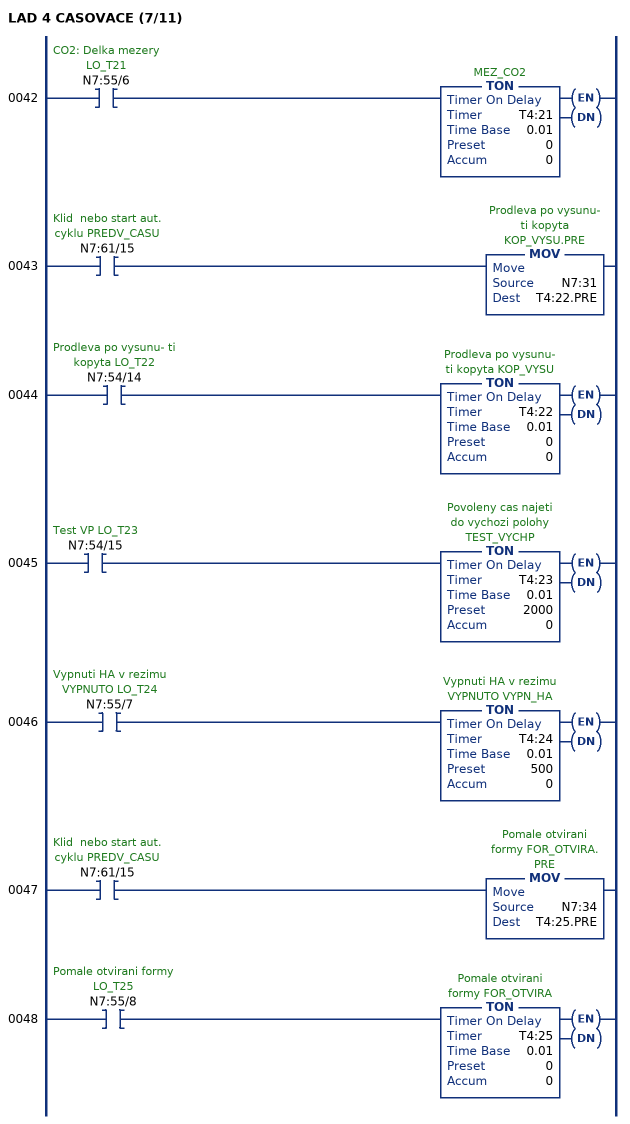
% Rung: 42 %
SOR XIC N7:55/6 TON T4:21 0.01 0 0 EOR
%   N7:55/6  LO_T21  "CO2: Delka mezery" %
%   T4:21  MEZ_CO2 %
% Rung: 43 %
SOR XIC N7:61/15 MOV N7:31 T4:22.PRE EOR
%   N7:61/15  PREDV_CASU  "Klid  nebo start aut. cyklu" %
%   N7:31  T_22  "Vysunut kopyto" %
%   T4:22  KOP_VYSU  "Prodleva po vysunu- ti kopyta" %
% Rung: 44 %
SOR XIC N7:54/14 TON T4:22 0.01 0 0 EOR
%   N7:54/14  LO_T22  "Prodleva po vysunu- ti kopyta" %
%   T4:22  KOP_VYSU  "Prodleva po vysunu- ti kopyta" %
% Rung: 45 %
SOR XIC N7:54/15 TON T4:23 0.01 2000 0 EOR
%   N7:54/15  LO_T23  "Test VP" %
%   T4:23  TEST_VYCHP  "Povoleny cas najeti do vychozi polohy" %
% Rung: 46 %
SOR XIC N7:55/7 TON T4:24 0.01 500 0 EOR
%   N7:55/7  LO_T24  "Vypnuti HA v rezimu VYPNUTO" %
%   T4:24  VYPN_HA  "Vypnuti HA v rezimu VYPNUTO" %
% Rung: 47 %
SOR XIC N7:61/15 MOV N7:34 T4:25.PRE EOR
%   N7:61/15  PREDV_CASU  "Klid  nebo start aut. cyklu" %
%   N7:34  T_25  "Otvrn formy pomalu" %
%   T4:25  FOR_OTVIRA  "Pomale otvirani formy" %
% Rung: 48 %
SOR XIC N7:55/8 TON T4:25 0.01 0 0 EOR
%   N7:55/8  LO_T25  "Pomale otvirani formy" %
%   T4:25  FOR_OTVIRA  "Pomale otvirani formy" %

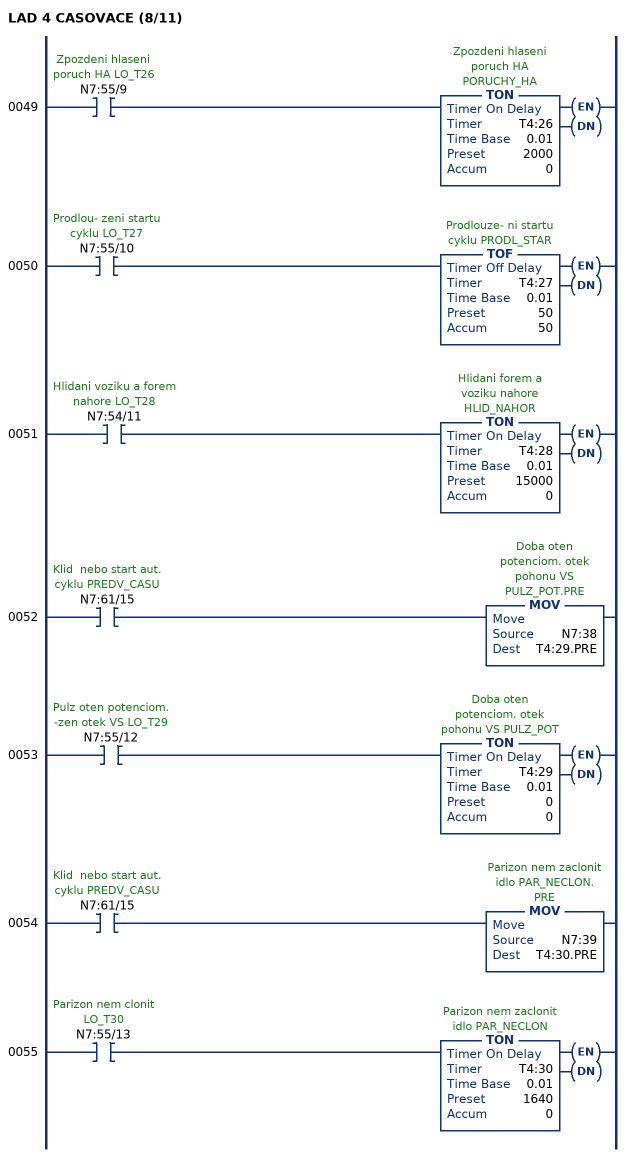
% Rung: 49 %
SOR XIC N7:55/9 TON T4:26 0.01 2000 0 EOR
%   N7:55/9  LO_T26  "Zpozdeni hlaseni poruch HA" %
%   T4:26  PORUCHY_HA  "Zpozdeni hlaseni poruch HA" %
% Rung: 50 %
SOR XIC N7:55/10 TOF T4:27 0.01 50 50 EOR
%   N7:55/10  LO_T27  "Prodlou- zeni startu cyklu" %
%   T4:27  PRODL_STAR  "Prodlouze- ni startu cyklu" %
% Rung: 51 %
SOR XIC N7:54/11 TON T4:28 0.01 15000 0 EOR
%   N7:54/11  LO_T28  "Hlidani voziku a forem nahore" %
%   T4:28  HLID_NAHOR  "Hlidani forem a voziku nahore" %
% Rung: 52 %
SOR XIC N7:61/15 MOV N7:38 T4:29.PRE EOR
%   N7:61/15  PREDV_CASU  "Klid  nebo start aut. cyklu" %
%   N7:38  T_29 %
%   T4:29  PULZ_POT  "Doba oten potenciom. otek pohonu VS" %
% Rung: 53 %
SOR XIC N7:55/12 TON T4:29 0.01 0 0 EOR
%   N7:55/12  LO_T29  "Pulz oten potenciom. -zen otek VS" %
%   T4:29  PULZ_POT  "Doba oten potenciom. otek pohonu VS" %
% Rung: 54 %
SOR XIC N7:61/15 MOV N7:39 T4:30.PRE EOR
%   N7:61/15  PREDV_CASU  "Klid  nebo start aut. cyklu" %
%   N7:39  T_30 %
%   T4:30  PAR_NECLON  "Parizon nem zaclonit idlo" %
% Rung: 55 %
SOR XIC N7:55/13 TON T4:30 0.01 1640 0 EOR
%   N7:55/13  LO_T30  "Parizon nem clonit" %
%   T4:30  PAR_NECLON  "Parizon nem zaclonit idlo" %

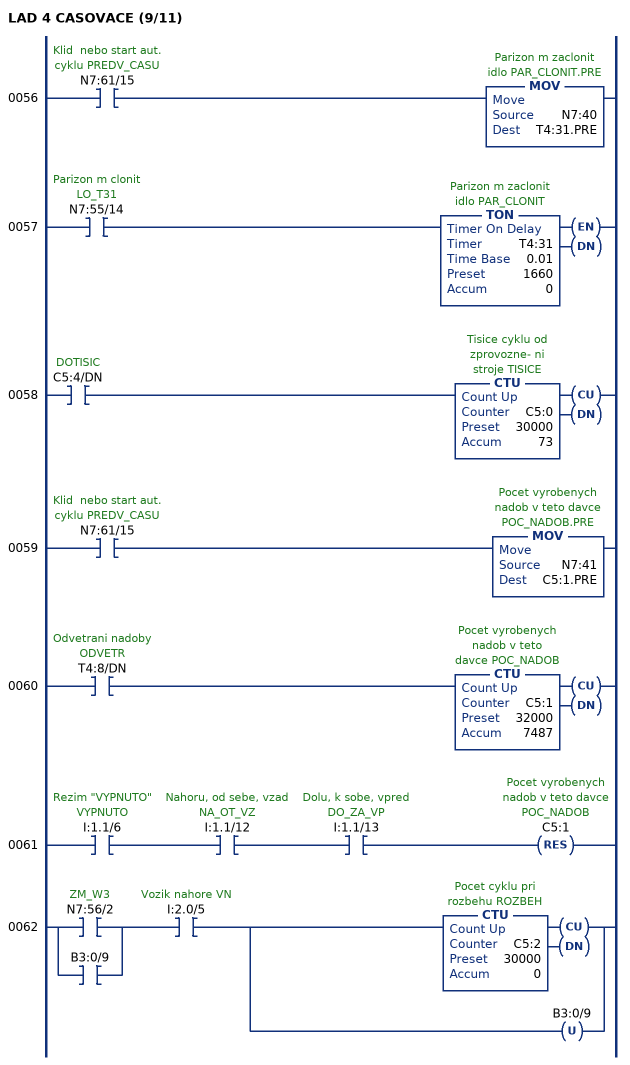
% Rung: 56 %
SOR XIC N7:61/15 MOV N7:40 T4:31.PRE EOR
%   N7:61/15  PREDV_CASU  "Klid  nebo start aut. cyklu" %
%   N7:40  T_31 %
%   T4:31  PAR_CLONIT  "Parizon m zaclonit idlo" %
% Rung: 57 %
SOR XIC N7:55/14 TON T4:31 0.01 1660 0 EOR
%   N7:55/14  LO_T31  "Parizon m clonit" %
%   T4:31  PAR_CLONIT  "Parizon m zaclonit idlo" %
% Rung: 58 %
SOR XIC C5:4/DN CTU C5:0 30000 73 EOR
%   C5:4/DN  DOTISIC %
%   C5:0  TISICE  "Tisice cyklu od zprovozne- ni stroje" %
% Rung: 59 %
SOR XIC N7:61/15 MOV N7:41 C5:1.PRE EOR
%   N7:61/15  PREDV_CASU  "Klid  nebo start aut. cyklu" %
%   N7:41  NADOBY_KS  "Pocet vyrobenych nadob" %
%   C5:1  POC_NADOB  "Pocet vyrobenych nadob v teto davce" %
% Rung: 60 %
SOR XIC T4:8/DN CTU C5:1 32000 7487 EOR
%   T4:8/DN  ODVETR  "Odvetrani nadoby" %
%   C5:1  POC_NADOB  "Pocet vyrobenych nadob v teto davce" %
% Rung: 61 %
SOR XIC I:1.1/6 XIC I:1.1/12 XIC I:1.1/13 RES C5:1 EOR
%   I:1.1/6  VYPNUTO  "Rezim "VYPNUTO"" %
%   I:1.1/12  NA_OT_VZ  "Nahoru, od sebe, vzad" %
%   I:1.1/13  DO_ZA_VP  "Dolu, k sobe, vpred" %
%   C5:1  POC_NADOB  "Pocet vyrobenych nadob v teto davce" %
% Rung: 62 %
SOR BST XIC N7:56/2 NXB XIC B3:0/9 BND XIC I:2.0/5 BST CTU C5:2 30000 0 NXB OTU B3:0/9 BND EOR
%   N7:56/2  ZM_W3 %
%   I:2.0/5  VN  "Vozik nahore" %
%   C5:2  ROZBEH  "Pocet cyklu pri rozbehu" %

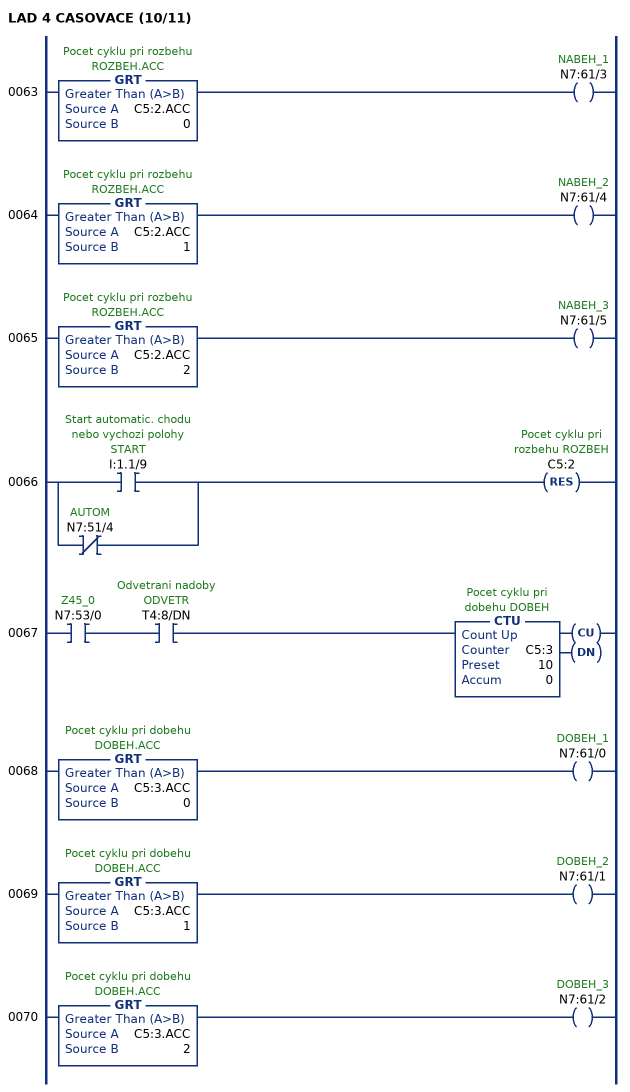
% Rung: 63 %
SOR GRT C5:2.ACC 0 OTE N7:61/3 EOR
%   C5:2  ROZBEH  "Pocet cyklu pri rozbehu" %
%   N7:61/3  NABEH_1 %
% Rung: 64 %
SOR GRT C5:2.ACC 1 OTE N7:61/4 EOR
%   C5:2  ROZBEH  "Pocet cyklu pri rozbehu" %
%   N7:61/4  NABEH_2 %
% Rung: 65 %
SOR GRT C5:2.ACC 2 OTE N7:61/5 EOR
%   C5:2  ROZBEH  "Pocet cyklu pri rozbehu" %
%   N7:61/5  NABEH_3 %
% Rung: 66 %
SOR BST XIC I:1.1/9 NXB XIO N7:51/4 BND RES C5:2 EOR
%   I:1.1/9  START  "Start automatic. chodu nebo vychozi polohy" %
%   N7:51/4  AUTOM %
%   C5:2  ROZBEH  "Pocet cyklu pri rozbehu" %
% Rung: 67 %
SOR XIC N7:53/0 XIC T4:8/DN CTU C5:3 10 0 EOR
%   N7:53/0  Z45_0 %
%   T4:8/DN  ODVETR  "Odvetrani nadoby" %
%   C5:3  DOBEH  "Pocet cyklu pri dobehu" %
% Rung: 68 %
SOR GRT C5:3.ACC 0 OTE N7:61/0 EOR
%   C5:3  DOBEH  "Pocet cyklu pri dobehu" %
%   N7:61/0  DOBEH_1 %
% Rung: 69 %
SOR GRT C5:3.ACC 1 OTE N7:61/1 EOR
%   C5:3  DOBEH  "Pocet cyklu pri dobehu" %
%   N7:61/1  DOBEH_2 %
% Rung: 70 %
SOR GRT C5:3.ACC 2 OTE N7:61/2 EOR
%   C5:3  DOBEH  "Pocet cyklu pri dobehu" %
%   N7:61/2  DOBEH_3 %

